TYPE ST_TrackConfig :
STRUCT
	TargetPosnBeforeTrackEnd	: LREAL := 100;
	StopPosPowermat				: LREAL := 7611;
END_STRUCT
END_TYPE

(* stored: Version 1.1.0.1
   DUT ST_TrackConfig: Id {0bf444be-035e-0e71-1156-30382b0847a6} *)
